{attribute addProperty BoxType "EJ4018-0000-0016"}
{attribute addProperty Id "AO_Outputs_ChannelAT %Q*ARRAY[0..7] OF AO_Outputs_Channel_F57FA4F9128160WcStateAT %I*WcState_28A8677510.1250InfoDataAT %I*InfoData_BC63D37F80100"}
{attribute addProperty CRC "220256351"}
{attribute addProperty SizeInBites "209"}
{attribute addProperty SizeInBytes "26.125"}
TYPE EJ4018_D5FA9EBB :
STRUCT
	{attribute addProperty Name "AO_Outputs_Channel"}
	AO_Outputs_Channel : ARRAY[0..7] OF AO_Outputs_Channel_F57FA4F9;
	{attribute addProperty Name "WcState"}
	WcState : WcState_28A86775;
	{attribute addProperty Name "InfoData"}
	InfoData : InfoData_BC63D37F;
END_STRUCT
END_TYPE

(* stored: Version 1.2.0.0, ProductVersion 3.1.4024.9
   DUT EJ4018_D5FA9EBB: Id {16b0fc56-e1b9-4ff4-b33b-755a1dd66afe} *)
